// TIA Portal V19 export
DATA_BLOCK "Peeler"   // DB63
// stored: InstanceOfName Peeler_FB, InstanceOfType FB
"Peeler_FB"
   // VAR_INPUT
   //    AreaInterface : "AreaInterface";
   //    ZSI : "udt_ZoneSafetyInterface";
   //    DSI : Struct
   //       LIft : "udt_DeviceSafetyInterface";
   //       Extension : "udt_DeviceSafetyInterface";
   //    END_STRUCT;
   //    DataIn : Struct
   //       Lift : "ValveMachine_DataIn";
   //       Extension : "ValveMachine_DataIn";
   //    END_STRUCT;
   //    CIn : Struct
   //       Manager : "Peeler_Manager";
   //       PressureRunning : Bool;
   //    END_STRUCT;
   //    Config : Struct
   //       Lift : "ValveMachine_Config";
   //       Extension : "ValveMachine_Config";
   //    END_STRUCT;
   // END_VAR
   // VAR_OUTPUT
   //    MachineInterface : "MachineInterface";
   //    DataOut : Struct
   //       Lift : "ValveMachine_DataOut";
   //       Extension : "ValveMachine_DataOut";
   //    END_STRUCT;
   //    COut : "Peeler_Status";
   // END_VAR
   // VAR
   //    Warning : Struct
   //       Lift { ExternalAccessible := 'False'; ExternalVisible := 'False'; ExternalWritable := 'False'} : "ValveMachine_Wng";
   //       Extension { ExternalAccessible := 'False'; ExternalVisible := 'False'; ExternalWritable := 'False'} : "ValveMachine_Wng";
   //    END_STRUCT;
   //    Alarm : Struct
   //       Lift : "ValveAlr";
   //       Extension : "ValveAlr";
   //    END_STRUCT;
   //    Sts : Struct
   //       dummy : Bool;
   //    END_STRUCT;
   //    Ctrl : Struct
   //       Move_Dwn_Aut : Bool;
   //       Move_Up_Aut : Bool;
   //    END_STRUCT;
   //    Lift : "ValveMachine_FB";
   //    Extension : "ValveMachine_FB";
   // END_VAR
BEGIN
END_DATA_BLOCK
